// TIA Portal V21 export
FUNCTION "LineAnimationFC" : Void   // FC311, LAD
{ S7_Optimized_Access := 'TRUE' }
// stored: AutoNumber false, SetENOAutomatically false
BEGIN

REGION Network 1: "LineAnimationDb"
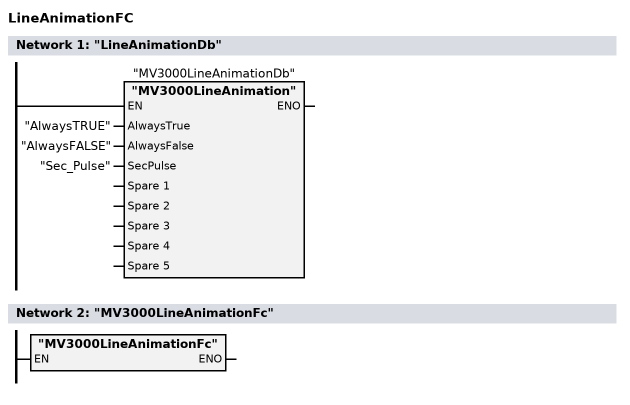
   RUNG wire#powerrail
      "MV3000LineAnimationDb"(AlwaysTrue := "AlwaysTRUE", AlwaysFalse := "AlwaysFALSE", SecPulse := "Sec_Pulse", "Spare 1" :=, "Spare 2" :=, "Spare 3" :=, "Spare 4" :=, "Spare 5" :=)
   END_RUNG
   // the same network as SCL:
   "MV3000LineAnimationDb"(AlwaysTrue := "AlwaysTRUE", AlwaysFalse := "AlwaysFALSE", SecPulse := "Sec_Pulse");   // "MV3000LineAnimation"
END_REGION

REGION Network 2: "MV3000LineAnimationFc"
   RUNG wire#powerrail
      "MV3000LineAnimationFc"()
   END_RUNG
   // the same network as SCL:
   "MV3000LineAnimationFc"();
END_REGION
END_FUNCTION
